Fanuc KAREL source: kt00894.KL

-- PROVISIONAL review KL for V940-1; original PC SHA256 f617030957dd2683aa8b8848be71da13dcb62ecc5524d68fa68f13b4a6e474b3
-- Incomplete behavior may be omitted. Consult companion uncertainty JSON. Do not deploy.
PROGRAM KT00894
%NOLOCKGROUP
VAR
  OUT : BOOLEAN
-- UNRESOLVED_DECL P1 type=000102
-- UNRESOLVED_DECL P2 type=000102
BEGIN
  -- V9_ZERO_TABLE_METADATA_HINT layout=0001; no indexed target words; source/name/runtime held
  -- UNRESOLVED_PC offsets 5-20; opcodes 2E,22,32,35
  -- UNRESOLVED_PC offsets 25-40; opcodes 2E,22,32,35
  -- UNRESOLVED_PC offsets 45-60; opcodes 2E,22,32,35
  -- UNRESOLVED_PC offsets 65-80; opcodes 2E,22,32,35
  -- UNRESOLVED_PC offsets 85-111; opcodes 27,27,49,7E,AD,27,9D,76,23
  -- UNRESOLVED_PC offsets 116-120; opcodes 7F
END KT00894
